ABB RAPID module: Module1.modx

MODULE Module1
    CONST robtarget HOLAHOLA:=[[309.74478014,345.099937686,96.09614673],[0.000000063,-0.000000086,0.923879543,0.382683407],[1,2,-2,0],[9E+09,9E+09,9E+09,9E+09,9E+09,9E+09]];
    CONST robtarget WidthPos:=[[40.536933297,176.929296343,945.886247295],[0.512837598,0.540603123,-0.468764624,-0.474347539],[1,-1,1,1],[9E+09,9E+09,9E+09,9E+09,9E+09,9E+09]];
    CONST robtarget Target_30:=[[-1531.934439138,0,0],[0.010403679,-0.026990672,0.004520625,0.999571324],[1,3,-1,1],[9E+09,9E+09,9E+09,9E+09,9E+09,9E+09]];
    CONST robtarget Target_20:=[[-590.986012171,0,0],[0.010403675,-0.026990699,0.004520689,0.999571323],[1,2,0,0],[9E+09,9E+09,9E+09,9E+09,9E+09,9E+09]];



ENDMODULE
